{attribute addProperty BoxType "EL1259-0000-0016"}
{attribute addProperty Id "CtrlAT %Q*Ctrl_ABBC220C678.3751OutputsAT %Q*Outputs_C23F921918623.2533Output_event_timeAT %Q*ARRAY[0 ..9] OF UDINT320400"}
{attribute addProperty CRC "787116963"}
{attribute addProperty SizeInBites "573"}
{attribute addProperty SizeInBytes "71.625"}
TYPE MTO_Outputs_10x_Channel_4C67AB5F :
STRUCT
	{attribute addProperty Name "Ctrl"}
	Ctrl AT %Q* : Ctrl_ABBC220C;
	{attribute addProperty Name "Outputs"}
	Outputs AT %Q* : Outputs_C23F9219;
	{attribute addProperty Name "Output_event_time"}
	Output_event_time AT %Q* : ARRAY[0 ..9] OF UDINT;
END_STRUCT
END_TYPE

(* stored: Version 1.2.0.0, ProductVersion 3.1.4024.9
   DUT MTO_Outputs_10x_Channel_4C67AB5F: Id {dc337037-3731-42e1-9bb7-363a359806f5} *)
